// ---- Tc3_DALI_PLC_Commissioning_Tool/VISUs/Visu_DALICommissioning/Visu_Part102Scenes.TcVIS
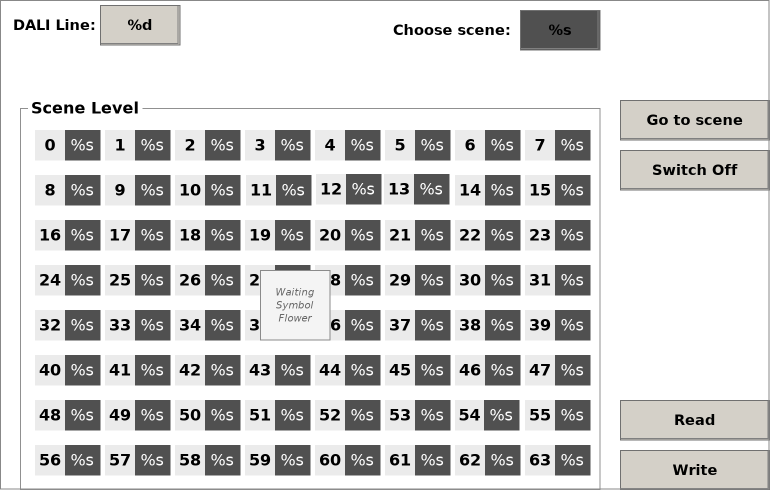
VISUALIZATION Visu_Part102Scenes  // 770x490
    GroupBox (20,100 580x390), "Scene Level"
        Group (85,30 65x30)
            Textfield (0,0 30x30), "1"
            Textfield (30,0 35x30), "%s", text variable: DALI_Commissioning.fbPart102Scenes.aScene[1], input disabled if: DALI_Commissioning.fbPart102Scenes.aNoShortAddress[1]
                p55702900: DALI_Commissioning.fbPart102Scenes.aFont[1]
                OnMouseClick: write the text variable via Default, min 0, max 255, title "Scene Value"
        Group (505,30 65x30)
            Textfield (0,0 30x30), "7"
            Textfield (30,0 35x30), "%s", text variable: DALI_Commissioning.fbPart102Scenes.aScene[7], input disabled if: DALI_Commissioning.fbPart102Scenes.aNoShortAddress[7]
                p55702900: DALI_Commissioning.fbPart102Scenes.aFont[7]
                OnMouseClick: write the text variable via Default, min 0, max 255, title "Scene Value"
        Group (435,30 65x30)
            Textfield (0,0 30x30), "6"
            Textfield (30,0 35x30), "%s", text variable: DALI_Commissioning.fbPart102Scenes.aScene[6], input disabled if: DALI_Commissioning.fbPart102Scenes.aNoShortAddress[6]
                p55702900: DALI_Commissioning.fbPart102Scenes.aFont[6]
                OnMouseClick: write the text variable via Default, min 0, max 255, title "Scene Value"
        Group (365,30 65x30)
            Textfield (0,0 30x30), "5"
            Textfield (30,0 35x30), "%s", text variable: DALI_Commissioning.fbPart102Scenes.aScene[5], input disabled if: DALI_Commissioning.fbPart102Scenes.aNoShortAddress[5]
                p55702900: DALI_Commissioning.fbPart102Scenes.aFont[5]
                OnMouseClick: write the text variable via Default, min 0, max 255, title "Scene Value"
        Group (295,30 65x30)
            Textfield (0,0 30x30), "4"
            Textfield (30,0 35x30), "%s", text variable: DALI_Commissioning.fbPart102Scenes.aScene[4], input disabled if: DALI_Commissioning.fbPart102Scenes.aNoShortAddress[4]
                p55702900: DALI_Commissioning.fbPart102Scenes.aFont[4]
                OnMouseClick: write the text variable via Default, min 0, max 255, title "Scene Value"
        Group (225,30 65x30)
            Textfield (0,0 30x30), "3"
            Textfield (30,0 35x30), "%s", text variable: DALI_Commissioning.fbPart102Scenes.aScene[3], input disabled if: DALI_Commissioning.fbPart102Scenes.aNoShortAddress[3]
                p55702900: DALI_Commissioning.fbPart102Scenes.aFont[3]
                OnMouseClick: write the text variable via Default, min 0, max 255, title "Scene Value"
        Group (155,30 65x30)
            Textfield (0,0 30x30), "2"
            Textfield (30,0 35x30), "%s", text variable: DALI_Commissioning.fbPart102Scenes.aScene[2], input disabled if: DALI_Commissioning.fbPart102Scenes.aNoShortAddress[2]
                p55702900: DALI_Commissioning.fbPart102Scenes.aFont[2]
                OnMouseClick: write the text variable via Default, min 0, max 255, title "Scene Value"
        Group (15,75 65x30)
            Textfield (0,0 30x30), "8"
            Textfield (30,0 35x30), "%s", text variable: DALI_Commissioning.fbPart102Scenes.aScene[8], input disabled if: DALI_Commissioning.fbPart102Scenes.aNoShortAddress[8]
                p55702900: DALI_Commissioning.fbPart102Scenes.aFont[8]
                OnMouseClick: write the text variable via Default, min 0, max 255, title "Scene Value"
        Group (15,120 65x30)
            Textfield (0,0 30x30), "16"
            Textfield (30,0 35x30), "%s", text variable: DALI_Commissioning.fbPart102Scenes.aScene[16], input disabled if: DALI_Commissioning.fbPart102Scenes.aNoShortAddress[16]
                p55702900: DALI_Commissioning.fbPart102Scenes.aFont[16]
                OnMouseClick: write the text variable via Default, min 0, max 255, title "Scene Value"
        Group (15,165 65x30)
            Textfield (0,0 30x30), "24"
            Textfield (30,0 35x30), "%s", text variable: DALI_Commissioning.fbPart102Scenes.aScene[24], input disabled if: DALI_Commissioning.fbPart102Scenes.aNoShortAddress[24]
                p55702900: DALI_Commissioning.fbPart102Scenes.aFont[24]
                OnMouseClick: write the text variable via Default, min 0, max 255, title "Scene Value"
        Group (15,210 65x30)
            Textfield (0,0 30x30), "32"
            Textfield (30,0 35x30), "%s", text variable: DALI_Commissioning.fbPart102Scenes.aScene[32], input disabled if: DALI_Commissioning.fbPart102Scenes.aNoShortAddress[32]
                p55702900: DALI_Commissioning.fbPart102Scenes.aFont[32]
                OnMouseClick: write the text variable via Default, min 0, max 255, title "Scene Value"
        Group (15,255 65x30)
            Textfield (0,0 30x30), "40"
            Textfield (30,0 35x30), "%s", text variable: DALI_Commissioning.fbPart102Scenes.aScene[40], input disabled if: DALI_Commissioning.fbPart102Scenes.aNoShortAddress[40]
                p55702900: DALI_Commissioning.fbPart102Scenes.aFont[40]
                OnMouseClick: write the text variable via Default, min 0, max 255, title "Scene Value"
        Group (15,300 65x30)
            Textfield (0,0 30x30), "48"
            Textfield (30,0 35x30), "%s", text variable: DALI_Commissioning.fbPart102Scenes.aScene[48], input disabled if: DALI_Commissioning.fbPart102Scenes.aNoShortAddress[48]
                p55702900: DALI_Commissioning.fbPart102Scenes.aFont[48]
                OnMouseClick: write the text variable via Default, min 0, max 255, title "Scene Value"
        Group (15,345 65x30)
            Textfield (0,0 30x30), "56"
            Textfield (30,0 35x30), "%s", text variable: DALI_Commissioning.fbPart102Scenes.aScene[56], input disabled if: DALI_Commissioning.fbPart102Scenes.aNoShortAddress[56]
                p55702900: DALI_Commissioning.fbPart102Scenes.aFont[56]
                OnMouseClick: write the text variable via Default, min 0, max 255, title "Scene Value"
        Group (85,75 65x30)
            Textfield (0,0 30x30), "9"
            Textfield (30,0 35x30), "%s", text variable: DALI_Commissioning.fbPart102Scenes.aScene[9], input disabled if: DALI_Commissioning.fbPart102Scenes.aNoShortAddress[9]
                p55702900: DALI_Commissioning.fbPart102Scenes.aFont[9]
                OnMouseClick: write the text variable via Default, min 0, max 255, title "Scene Value"
        Group (155,75 65x30)
            Textfield (0,0 30x30), "10"
            Textfield (30,0 35x30), "%s", text variable: DALI_Commissioning.fbPart102Scenes.aScene[10], input disabled if: DALI_Commissioning.fbPart102Scenes.aNoShortAddress[10]
                p55702900: DALI_Commissioning.fbPart102Scenes.aFont[10]
                OnMouseClick: write the text variable via Default, min 0, max 255, title "Scene Value"
        Group (226,75 65x30)
            Textfield (0,0 30x30), "11"
            Textfield (30,0 35x30), "%s", text variable: DALI_Commissioning.fbPart102Scenes.aScene[11], input disabled if: DALI_Commissioning.fbPart102Scenes.aNoShortAddress[11]
                p55702900: DALI_Commissioning.fbPart102Scenes.aFont[11]
                OnMouseClick: write the text variable via Default, min 0, max 255, title "Scene Value"
        Group (296,74 65x30)
            Textfield (0,0 30x30), "12"
            Textfield (30,0 35x30), "%s", text variable: DALI_Commissioning.fbPart102Scenes.aScene[12], input disabled if: DALI_Commissioning.fbPart102Scenes.aNoShortAddress[12]
                p55702900: DALI_Commissioning.fbPart102Scenes.aFont[12]
                OnMouseClick: write the text variable via Default, min 0, max 255, title "Scene Value"
        Group (364,74 65x30)
            Textfield (0,0 30x30), "13"
            Textfield (30,0 35x30), "%s", text variable: DALI_Commissioning.fbPart102Scenes.aScene[13], input disabled if: DALI_Commissioning.fbPart102Scenes.aNoShortAddress[13]
                p55702900: DALI_Commissioning.fbPart102Scenes.aFont[13]
                OnMouseClick: write the text variable via Default, min 0, max 255, title "Scene Value"
        Group (435,75 65x30)
            Textfield (0,0 30x30), "14"
            Textfield (30,0 35x30), "%s", text variable: DALI_Commissioning.fbPart102Scenes.aScene[14], input disabled if: DALI_Commissioning.fbPart102Scenes.aNoShortAddress[14]
                p55702900: DALI_Commissioning.fbPart102Scenes.aFont[14]
                OnMouseClick: write the text variable via Default, min 0, max 255, title "Scene Value"
        Group (505,75 65x30)
            Textfield (0,0 30x30), "15"
            Textfield (30,0 35x30), "%s", text variable: DALI_Commissioning.fbPart102Scenes.aScene[15], input disabled if: DALI_Commissioning.fbPart102Scenes.aNoShortAddress[15]
                p55702900: DALI_Commissioning.fbPart102Scenes.aFont[15]
                OnMouseClick: write the text variable via Default, min 0, max 255, title "Scene Value"
        Group (85,120 65x30)
            Textfield (0,0 30x30), "17"
            Textfield (30,0 35x30), "%s", text variable: DALI_Commissioning.fbPart102Scenes.aScene[17], input disabled if: DALI_Commissioning.fbPart102Scenes.aNoShortAddress[17]
                p55702900: DALI_Commissioning.fbPart102Scenes.aFont[17]
                OnMouseClick: write the text variable via Default, min 0, max 255, title "Scene Value"
        Group (155,120 65x30)
            Textfield (0,0 30x30), "18"
            Textfield (30,0 35x30), "%s", text variable: DALI_Commissioning.fbPart102Scenes.aScene[18], input disabled if: DALI_Commissioning.fbPart102Scenes.aNoShortAddress[18]
                p55702900: DALI_Commissioning.fbPart102Scenes.aFont[18]
                OnMouseClick: write the text variable via Default, min 0, max 255, title "Scene Value"
        Group (225,120 65x30)
            Textfield (0,0 30x30), "19"
            Textfield (30,0 35x30), "%s", text variable: DALI_Commissioning.fbPart102Scenes.aScene[19], input disabled if: DALI_Commissioning.fbPart102Scenes.aNoShortAddress[19]
                p55702900: DALI_Commissioning.fbPart102Scenes.aFont[19]
                OnMouseClick: write the text variable via Default, min 0, max 255, title "Scene Value"
        Group (295,120 65x30)
            Textfield (0,0 30x30), "20"
            Textfield (30,0 35x30), "%s", text variable: DALI_Commissioning.fbPart102Scenes.aScene[20], input disabled if: DALI_Commissioning.fbPart102Scenes.aNoShortAddress[20]
                p55702900: DALI_Commissioning.fbPart102Scenes.aFont[20]
                OnMouseClick: write the text variable via Default, min 0, max 255, title "Scene Value"
        Group (365,120 65x30)
            Textfield (0,0 30x30), "21"
            Textfield (30,0 35x30), "%s", text variable: DALI_Commissioning.fbPart102Scenes.aScene[21], input disabled if: DALI_Commissioning.fbPart102Scenes.aNoShortAddress[21]
                p55702900: DALI_Commissioning.fbPart102Scenes.aFont[21]
                OnMouseClick: write the text variable via Default, min 0, max 255, title "Scene Value"
        Group (435,120 65x30)
            Textfield (0,0 30x30), "22"
            Textfield (30,0 35x30), "%s", text variable: DALI_Commissioning.fbPart102Scenes.aScene[22], input disabled if: DALI_Commissioning.fbPart102Scenes.aNoShortAddress[22]
                p55702900: DALI_Commissioning.fbPart102Scenes.aFont[22]
                OnMouseClick: write the text variable via Default, min 0, max 255, title "Scene Value"
        Group (505,120 65x30)
            Textfield (0,0 30x30), "23"
            Textfield (30,0 35x30), "%s", text variable: DALI_Commissioning.fbPart102Scenes.aScene[23], input disabled if: DALI_Commissioning.fbPart102Scenes.aNoShortAddress[23]
                p55702900: DALI_Commissioning.fbPart102Scenes.aFont[23]
                OnMouseClick: write the text variable via Default, min 0, max 255, title "Scene Value"
        Group (85,165 65x30)
            Textfield (0,0 30x30), "25"
            Textfield (30,0 35x30), "%s", text variable: DALI_Commissioning.fbPart102Scenes.aScene[25], input disabled if: DALI_Commissioning.fbPart102Scenes.aNoShortAddress[25]
                p55702900: DALI_Commissioning.fbPart102Scenes.aFont[25]
                OnMouseClick: write the text variable via Default, min 0, max 255, title "Scene Value"
        Group (155,165 65x30)
            Textfield (0,0 30x30), "26"
            Textfield (30,0 35x30), "%s", text variable: DALI_Commissioning.fbPart102Scenes.aScene[26], input disabled if: DALI_Commissioning.fbPart102Scenes.aNoShortAddress[26]
                p55702900: DALI_Commissioning.fbPart102Scenes.aFont[26]
                OnMouseClick: write the text variable via Default, min 0, max 255, title "Scene Value"
        Group (225,165 65x30)
            Textfield (0,0 30x30), "27"
            Textfield (30,0 35x30), "%s", text variable: DALI_Commissioning.fbPart102Scenes.aScene[27], input disabled if: DALI_Commissioning.fbPart102Scenes.aNoShortAddress[27]
                p55702900: DALI_Commissioning.fbPart102Scenes.aFont[27]
                OnMouseClick: write the text variable via Default, min 0, max 255, title "Scene Value"
        Group (295,165 65x30)
            Textfield (0,0 30x30), "28"
            Textfield (30,0 35x30), "%s", text variable: DALI_Commissioning.fbPart102Scenes.aScene[28], input disabled if: DALI_Commissioning.fbPart102Scenes.aNoShortAddress[28]
                p55702900: DALI_Commissioning.fbPart102Scenes.aFont[28]
                OnMouseClick: write the text variable via Default, min 0, max 255, title "Scene Value"
        Group (365,165 65x30)
            Textfield (0,0 30x30), "29"
            Textfield (30,0 35x30), "%s", text variable: DALI_Commissioning.fbPart102Scenes.aScene[29], input disabled if: DALI_Commissioning.fbPart102Scenes.aNoShortAddress[29]
                p55702900: DALI_Commissioning.fbPart102Scenes.aFont[29]
                OnMouseClick: write the text variable via Default, min 0, max 255, title "Scene Value"
        Group (435,165 65x30)
            Textfield (0,0 30x30), "30"
            Textfield (30,0 35x30), "%s", text variable: DALI_Commissioning.fbPart102Scenes.aScene[30], input disabled if: DALI_Commissioning.fbPart102Scenes.aNoShortAddress[30]
                p55702900: DALI_Commissioning.fbPart102Scenes.aFont[30]
                OnMouseClick: write the text variable via Default, min 0, max 255, title "Scene Value"
        Group (505,165 65x30)
            Textfield (0,0 30x30), "31"
            Textfield (30,0 35x30), "%s", text variable: DALI_Commissioning.fbPart102Scenes.aScene[31], input disabled if: DALI_Commissioning.fbPart102Scenes.aNoShortAddress[31]
                p55702900: DALI_Commissioning.fbPart102Scenes.aFont[31]
                OnMouseClick: write the text variable via Default, min 0, max 255, title "Scene Value"
        Group (85,210 65x30)
            Textfield (0,0 30x30), "33"
            Textfield (30,0 35x30), "%s", text variable: DALI_Commissioning.fbPart102Scenes.aScene[33], input disabled if: DALI_Commissioning.fbPart102Scenes.aNoShortAddress[32]
                p55702900: DALI_Commissioning.fbPart102Scenes.aFont[33]
                OnMouseClick: write the text variable via Default, min 0, max 255, title "Scene Value"
        Group (155,210 65x30)
            Textfield (0,0 30x30), "34"
            Textfield (30,0 35x30), "%s", text variable: DALI_Commissioning.fbPart102Scenes.aScene[34], input disabled if: DALI_Commissioning.fbPart102Scenes.aNoShortAddress[34]
                p55702900: DALI_Commissioning.fbPart102Scenes.aFont[34]
                OnMouseClick: write the text variable via Default, min 0, max 255, title "Scene Value"
        Group (295,210 65x30)
            Textfield (0,0 30x30), "36"
            Textfield (30,0 35x30), "%s", text variable: DALI_Commissioning.fbPart102Scenes.aScene[36], input disabled if: DALI_Commissioning.fbPart102Scenes.aNoShortAddress[36]
                p55702900: DALI_Commissioning.fbPart102Scenes.aFont[36]
                OnMouseClick: write the text variable via Default, min 0, max 255
        Group (365,210 65x30)
            Textfield (0,0 30x30), "37"
            Textfield (30,0 35x30), "%s", text variable: DALI_Commissioning.fbPart102Scenes.aScene[37], input disabled if: DALI_Commissioning.fbPart102Scenes.aNoShortAddress[37]
                p55702900: DALI_Commissioning.fbPart102Scenes.aFont[37]
                OnMouseClick: write the text variable via Default, min 0, max 255, title "Scene Value"
        Group (435,210 65x30)
            Textfield (0,0 30x30), "38"
            Textfield (30,0 35x30), "%s", text variable: DALI_Commissioning.fbPart102Scenes.aScene[38], input disabled if: DALI_Commissioning.fbPart102Scenes.aNoShortAddress[38]
                p55702900: DALI_Commissioning.fbPart102Scenes.aFont[38]
                OnMouseClick: write the text variable via Default, min 0, max 255, title "Scene Value"
        Group (505,210 65x30)
            Textfield (0,0 30x30), "39"
            Textfield (30,0 35x30), "%s", text variable: DALI_Commissioning.fbPart102Scenes.aScene[39], input disabled if: DALI_Commissioning.fbPart102Scenes.aNoShortAddress[39]
                p55702900: DALI_Commissioning.fbPart102Scenes.aFont[39]
                OnMouseClick: write the text variable via Default, min 0, max 255, title "Scene Value"
        Group (85,255 65x30)
            Textfield (0,0 30x30), "41"
            Textfield (30,0 35x30), "%s", text variable: DALI_Commissioning.fbPart102Scenes.aScene[41], input disabled if: DALI_Commissioning.fbPart102Scenes.aNoShortAddress[41]
                p55702900: DALI_Commissioning.fbPart102Scenes.aFont[41]
                OnMouseClick: write the text variable via Default, min 0, max 255, title "Scene Value"
        Group (155,255 65x30)
            Textfield (0,0 30x30), "42"
            Textfield (30,0 35x30), "%s", text variable: DALI_Commissioning.fbPart102Scenes.aScene[42], input disabled if: DALI_Commissioning.fbPart102Scenes.aNoShortAddress[42]
                p55702900: DALI_Commissioning.fbPart102Scenes.aFont[42]
                OnMouseClick: write the text variable via Default, min 0, max 255, title "Scene Value"
        Group (225,210 65x30)
            Textfield (0,0 30x30), "35"
            Textfield (30,0 35x30), "%s", text variable: DALI_Commissioning.fbPart102Scenes.aScene[35], input disabled if: DALI_Commissioning.fbPart102Scenes.aNoShortAddress[35]
                p55702900: DALI_Commissioning.fbPart102Scenes.aFont[35]
                OnMouseClick: write the text variable via Default, min 0, max 255, title "Scene Value"
        Group (225,255 65x30)
            Textfield (0,0 30x30), "43"
            Textfield (30,0 35x30), "%s", text variable: DALI_Commissioning.fbPart102Scenes.aScene[43], input disabled if: DALI_Commissioning.fbPart102Scenes.aNoShortAddress[43]
                p55702900: DALI_Commissioning.fbPart102Scenes.aFont[43]
                OnMouseClick: write the text variable via Default, min 0, max 255, title "Scene Value"
        Group (295,255 65x30)
            Textfield (0,0 30x30), "44"
            Textfield (30,0 35x30), "%s", text variable: DALI_Commissioning.fbPart102Scenes.aScene[44], input disabled if: DALI_Commissioning.fbPart102Scenes.aNoShortAddress[44]
                p55702900: DALI_Commissioning.fbPart102Scenes.aFont[44]
                OnMouseClick: write the text variable via Default, min 0, max 255, title "Scene Value"
        Group (365,255 65x30)
            Textfield (0,0 30x30), "45"
            Textfield (30,0 35x30), "%s", text variable: DALI_Commissioning.fbPart102Scenes.aScene[45], input disabled if: DALI_Commissioning.fbPart102Scenes.aNoShortAddress[45]
                p55702900: DALI_Commissioning.fbPart102Scenes.aFont[45]
                OnMouseClick: write the text variable via Default, min 0, max 255, title "Scene Value"
        Group (435,255 65x30)
            Textfield (0,0 30x30), "46"
            Textfield (30,0 35x30), "%s", text variable: DALI_Commissioning.fbPart102Scenes.aScene[46], input disabled if: DALI_Commissioning.fbPart102Scenes.aNoShortAddress[46]
                p55702900: DALI_Commissioning.fbPart102Scenes.aFont[46]
                OnMouseClick: write the text variable via Default, min 0, max 255, title "Scene Value"
        Group (505,255 65x30)
            Textfield (0,0 30x30), "47"
            Textfield (30,0 35x30), "%s", text variable: DALI_Commissioning.fbPart102Scenes.aScene[47], input disabled if: DALI_Commissioning.fbPart102Scenes.aNoShortAddress[47]
                p55702900: DALI_Commissioning.fbPart102Scenes.aFont[47]
                OnMouseClick: write the text variable via Default, min 0, max 255, title "Scene Value"
        Group (85,300 65x30)
            Textfield (0,0 30x30), "49"
            Textfield (30,0 35x30), "%s", text variable: DALI_Commissioning.fbPart102Scenes.aScene[49], input disabled if: DALI_Commissioning.fbPart102Scenes.aNoShortAddress[49]
                p55702900: DALI_Commissioning.fbPart102Scenes.aFont[49]
                OnMouseClick: write the text variable via Default, min 0, max 255, title "Scene Value"
        Group (155,300 65x30)
            Textfield (0,0 30x30), "50"
            Textfield (30,0 35x30), "%s", text variable: DALI_Commissioning.fbPart102Scenes.aScene[50], input disabled if: DALI_Commissioning.fbPart102Scenes.aNoShortAddress[50]
                p55702900: DALI_Commissioning.fbPart102Scenes.aFont[50]
                OnMouseClick: write the text variable via Default, min 0, max 255, title "Scene Value"
        Group (225,300 65x30)
            Textfield (0,0 30x30), "51"
            Textfield (30,0 35x30), "%s", text variable: DALI_Commissioning.fbPart102Scenes.aScene[51], input disabled if: DALI_Commissioning.fbPart102Scenes.aNoShortAddress[51]
                p55702900: DALI_Commissioning.fbPart102Scenes.aFont[51]
                OnMouseClick: write the text variable via Default, min 0, max 255, title "Scene Value"
        Group (295,300 65x30)
            Textfield (0,0 30x30), "52"
            Textfield (30,0 35x30), "%s", text variable: DALI_Commissioning.fbPart102Scenes.aScene[52], input disabled if: DALI_Commissioning.fbPart102Scenes.aNoShortAddress[52]
                p55702900: DALI_Commissioning.fbPart102Scenes.aFont[52]
                OnMouseClick: write the text variable via Default, min 0, max 255, title "Scene Value"
        Group (365,300 65x30)
            Textfield (0,0 30x30), "53"
            Textfield (30,0 35x30), "%s", text variable: DALI_Commissioning.fbPart102Scenes.aScene[53], input disabled if: DALI_Commissioning.fbPart102Scenes.aNoShortAddress[53]
                p55702900: DALI_Commissioning.fbPart102Scenes.aFont[53]
                OnMouseClick: write the text variable via Default, min 0, max 255, title "Scene Value"
        Group (435,300 64x30)
            Textfield (0,0 29x30), "54"
            Textfield (29,0 35x30), "%s", text variable: DALI_Commissioning.fbPart102Scenes.aScene[54], input disabled if: DALI_Commissioning.fbPart102Scenes.aNoShortAddress[54]
                p55702900: DALI_Commissioning.fbPart102Scenes.aFont[54]
                OnMouseClick: write the text variable via Default, min 0, max 255, title "Scene Value"
        Group (505,300 65x30)
            Textfield (0,0 30x30), "55"
            Textfield (30,0 35x30), "%s", text variable: DALI_Commissioning.fbPart102Scenes.aScene[55], input disabled if: DALI_Commissioning.fbPart102Scenes.aNoShortAddress[55]
                p55702900: DALI_Commissioning.fbPart102Scenes.aFont[55]
                OnMouseClick: write the text variable via Default, min 0, max 255, title "Scene Value"
        Group (85,345 65x30)
            Textfield (0,0 30x30), "57"
            Textfield (30,0 35x30), "%s", text variable: DALI_Commissioning.fbPart102Scenes.aScene[57], input disabled if: DALI_Commissioning.fbPart102Scenes.aNoShortAddress[57]
                p55702900: DALI_Commissioning.fbPart102Scenes.aFont[57]
                OnMouseClick: write the text variable via Default, min 0, max 255, title "Scene Value"
        Group (155,345 65x30)
            Textfield (0,0 30x30), "58"
            Textfield (30,0 35x30), "%s", text variable: DALI_Commissioning.fbPart102Scenes.aScene[58], input disabled if: DALI_Commissioning.fbPart102Scenes.aNoShortAddress[58]
                p55702900: DALI_Commissioning.fbPart102Scenes.aFont[58]
                OnMouseClick: write the text variable via Default, min 0, max 255, title "Scene Value"
        Group (225,345 65x30)
            Textfield (0,0 30x30), "59"
            Textfield (30,0 35x30), "%s", text variable: DALI_Commissioning.fbPart102Scenes.aScene[59], input disabled if: DALI_Commissioning.fbPart102Scenes.aNoShortAddress[59]
                p55702900: DALI_Commissioning.fbPart102Scenes.aFont[59]
                OnMouseClick: write the text variable via Default, min 0, max 255, title "Scene Value"
        Group (295,345 65x30)
            Textfield (0,0 30x30), "60"
            Textfield (30,0 35x30), "%s", text variable: DALI_Commissioning.fbPart102Scenes.aScene[60], input disabled if: DALI_Commissioning.fbPart102Scenes.aNoShortAddress[60]
                p55702900: DALI_Commissioning.fbPart102Scenes.aFont[60]
                OnMouseClick: write the text variable via Default, min 0, max 255, title "Scene Value"
        Group (365,345 65x30)
            Textfield (0,0 30x30), "61"
            Textfield (30,0 35x30), "%s", text variable: DALI_Commissioning.fbPart102Scenes.aScene[61], input disabled if: DALI_Commissioning.fbPart102Scenes.aNoShortAddress[61]
                p55702900: DALI_Commissioning.fbPart102Scenes.aFont[61]
                OnMouseClick: write the text variable via Default, min 0, max 255, title "Scene Value"
        Group (435,345 65x30)
            Textfield (0,0 30x30), "62"
            Textfield (30,0 35x30), "%s", text variable: DALI_Commissioning.fbPart102Scenes.aScene[62], input disabled if: DALI_Commissioning.fbPart102Scenes.aNoShortAddress[62]
                p55702900: DALI_Commissioning.fbPart102Scenes.aFont[62]
                OnMouseClick: write the text variable via Default, min 0, max 255, title "Scene Value"
        Group (505,345 65x30)
            Textfield (0,0 30x30), "63"
            Textfield (30,0 35x30), "%s", text variable: DALI_Commissioning.fbPart102Scenes.aScene[63], input disabled if: DALI_Commissioning.fbPart102Scenes.aNoShortAddress[63]
                p55702900: DALI_Commissioning.fbPart102Scenes.aFont[63]
                OnMouseClick: write the text variable via Default, min 0, max 255, title "Scene Value"
        WaitingSymbolFlower (240,170 70x70), invisible if: DALI_Commissioning.fbPart102Scenes.bHideWaitSymbol
        Group (15,30 65x30)
            Textfield (0,0 30x30), "0"
            Textfield (30,0 35x30), "%s", text variable: DALI_Commissioning.fbPart102Scenes.aScene[0], input disabled if: DALI_Commissioning.fbPart102Scenes.aNoShortAddress[0]
                p55702900: DALI_Commissioning.fbPart102Scenes.aFont[0]
                OnMouseClick: write the text variable via Default, min 0, max 255, title "Scene Value"
    Button (620,400 150x40), "Read"
        OnMouseClick: execute { DALI_Commissioning.fbPart102Scenes.bRead := TRUE; }
    Button (620,450 150x40), "Write"
        OnMouseClick: execute { DALI_Commissioning.fbPart102Scenes.bWrite := TRUE; }
    Button (620,100 150x40), "Go to scene"
        OnMouseClick: execute { DALI_Commissioning.fbPart102Scenes.bGoToScene := TRUE; }
    Button (620,150 150x40), "Switch Off"
        OnMouseClick: execute { DALI_Commissioning.fbPart102Scenes.bSwitchOff := TRUE; }
    Textfield (390,10 120x40), "Choose scene:"
    Button (520,10 80x40), "%s", text variable: DALI_Commissioning.fbPart102Scenes.nScene
        OnMouseClick: write the text variable via Default, min 0, max 15, title "Choose scene"
    Group (10,5 170x40)
        Textfield (0,0 110x40), "DALI Line:"
        Button (90,0 80x40), "%d", text variable: GVL_Internal.nDALILine
            OnMouseClick: write the text variable via Default, min 1, max GVL_Internal.nNumberOfDALI_Lines, title "Choose line"
END_VISUALIZATION

// ---- Tc3_DALI_PLC_Commissioning_Tool/VISUs/Visu_DALICommissioning/Visu_Part102SetFading.TcVIS
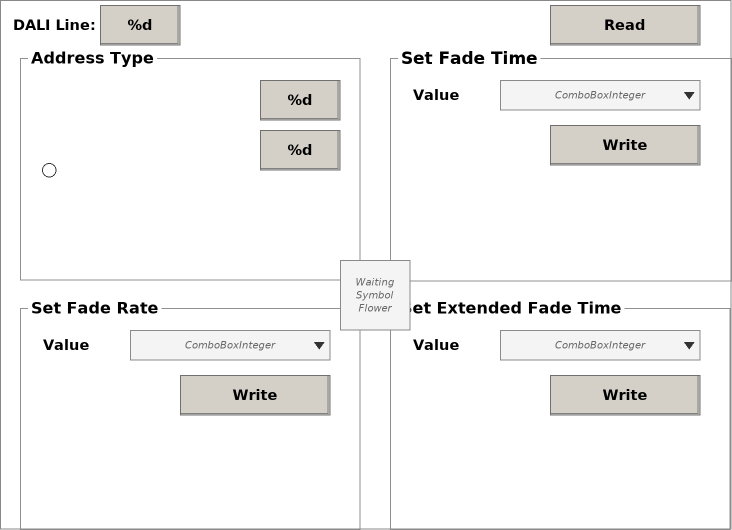
VISUALIZATION Visu_Part102SetFading  // 732x530
    GroupBox (390,50 342x231), "Set Fade Time"
        Textfield (20,30 100x30), "Value"
        ComboBoxInteger (110,30 200x30), variable: DALI_Commissioning.fbPart102SetFading.eFadeTime, text list: 'FadeTime'
        Button (160,75 150x40), "Write"
            OnMouseClick: execute { DALI_Commissioning.fbPart102SetFading.bWriteFadeTime := TRUE; }
    GroupBox (20,50 340x230), "Address Type"
        Button (240,30 80x40), "%d", text variable: DALI_Commissioning.fbPart102SetFading.nShortAddress
            OnMouseClick: write the text variable via Default, min 0, max 63, title "Insert Short Address"
        RadioButton (20,20 190x200), variable: DALI_Commissioning.fbPart102SetFading.eAddressType
            Areas[0]: Text=Short Address
            Areas[1]: Text=Group Address
            Areas[2]: Text=Broadcast
            Areas[3]: Text=Unaddressed
        Button (240,80 80x40), "%d", text variable: DALI_Commissioning.fbPart102SetFading.nGroupAddress
            OnMouseClick: write the text variable via Default, min 0, max 15, title "Insert Group Address"
    GroupBox (20,300 340x230), "Set Fade Rate"
        Textfield (20,30 100x30), "Value"
        ComboBoxInteger (110,30 200x30), variable: DALI_Commissioning.fbPart102SetFading.eFadeRate, text list: 'FadeRate'
        Button (160,75 150x40), "Write"
            OnMouseClick: execute { DALI_Commissioning.fbPart102setFading.bWriteFadeRate := TRUE; }
    GroupBox (390,300 340x230), "Set Extended Fade Time"
        Textfield (20,30 100x30), "Value"
        ComboBoxInteger (110,30 200x30), tooltip "Extended Fade Time only valid if Fade Time equals 0!", variable: DALI_Commissioning.fbPart102SetFading.eExtendedFadeTime, input disabled if: DALI_Commissioning.fbPart102SetFading.bNoFadeTime, text list: 'ExtendedFadeTime'
        Button (160,75 150x40), "Write", tooltip "Extended Fade Time only valid if Fade Time equals 0!", invisible if: DALI_Commissioning.fbPart102SetFading.bNoFadeTime, input disabled if: DALI_Commissioning.fbPart102SetFading.bNoFadeTime
            OnMouseClick: execute { DALI_Commissioning.fbPart102SetFading.bWriteExtendedFadeTime:=true; }
    Button (550,5 150x40), "Read", tooltip "Reads all Fading Parameters", invisible if: ( DALI_Commissioning.fbPart102SetFading.eAddressType >=1), input disabled if: ( DALI_Commissioning.fbPart102SetFading.eAddressType >=1)
        OnMouseClick: execute { DALI_Commissioning.fbPart102SetFading.bRead := TRUE; }
    WaitingSymbolFlower (340,260 70x70), invisible if: DALI_Commissioning.fbPart102SetFading.bHideWaitSymbol
    Group (10,5 170x40)
        Textfield (0,0 110x40), "DALI Line:"
        Button (90,0 80x40), "%d", text variable: GVL_Internal.nDALILine
            OnMouseClick: write the text variable via Default, min 1, max GVL_Internal.nNumberOfDALI_Lines, title "Choose line"
END_VISUALIZATION

// ---- Tc3_DALI_PLC_Commissioning_Tool/VISUs/Visu_DALICommissioning/Visu_Part103Addressing.TcVIS
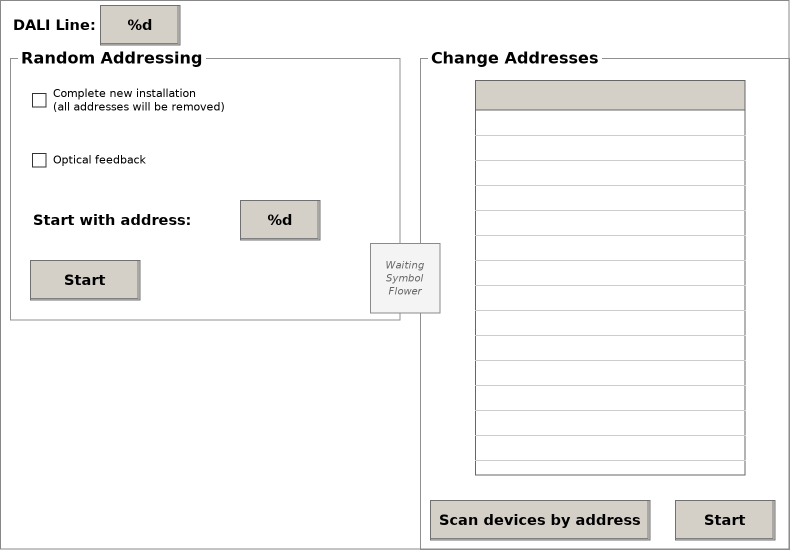
VISUALIZATION Visu_Part103Addressing  // 790x550
    GroupBox (420,50 370x500), "Change Addresses"
        Table (55,30 270x395), data array: DALI_Commissioning.fbPart103Addressing.aChangeAddressList
            p3854506369: DALI_Commissioning.fbPart103Addressing.aChangeAddressList[INDEX].nOldAddress
            p1892666644: DALI_Commissioning.fbPart103Addressing.aChangeAddressList[INDEX].nNewAddress
            p338671338: DALI_Commissioning.fbPart103Addressing.aChangeAddressList[INDEX].nRandomAddress
            p2170511999: DALI_Commissioning.fbPart103Addressing.aChangeAddressList[INDEX].nErrors
            Columns.Column.[0].Template: DALI_Commissioning.fbPart103Addressing.aNoShortAddress[INDEX]
            Columns.Column.[1].Template: DALI_Commissioning.fbPart103Addressing.aNoShortAddress[INDEX]; OnMouseClick: write the text variable via Default, min 0, max 63, title "New Short Address"
        Button (255,450 100x40), "Start"
            OnMouseClick: execute { DALI_Commissioning.fbPart103Addressing.bStartChangeAddress := TRUE; }
        Button (10,450 220x40), "Scan devices by address"
            OnMouseClick: execute { DALI_Commissioning.fbPart103Addressing.bScanDevices := TRUE; }
    GroupBox (10,50 390x270), "Random Addressing"
        Button (20,210 110x40), "Start"
            OnMouseClick: execute { DALI_Commissioning.fbPart103Addressing.bStartRandomAddressing := TRUE; }
        Checkbox (20,30 360x40), "Complete new installation (all addresses will be removed)", variable: DALI_Commissioning.fbPart103Addressing.bNewInstallation
        Checkbox (20,90 360x40), "Optical feedback", variable: DALI_Commissioning.fbPart103Addressing.bOpticalFeedback
        Textfield (20,150 200x40), "Start with address:"
        Button (230,150 80x40), "%d", text variable: DALI_Commissioning.fbPart103Addressing.nStartAddress
            OnMouseClick: write DALI_Commissioning.fbPart103Addressing.nStartAddress via Default, min 0, max 63, title "Insert Short Address"
    WaitingSymbolFlower (370,243 70x70), invisible if: DALI_Commissioning.fbPart103Addressing.bHideWaitSymbol
    Group (10,5 170x40)
        Textfield (0,0 110x40), "DALI Line:"
        Button (90,0 80x40), "%d", text variable: GVL_Internal.nDALILine
            OnMouseClick: write the text variable via Default, min 1, max GVL_Internal.nNumberOfDALI_Lines, title "Choose line"
END_VISUALIZATION

// ---- Tc3_DALI_PLC_Commissioning_Tool/VISUs/Visu_DALICommissioning/Visu_Part103MemoryBank.TcVIS
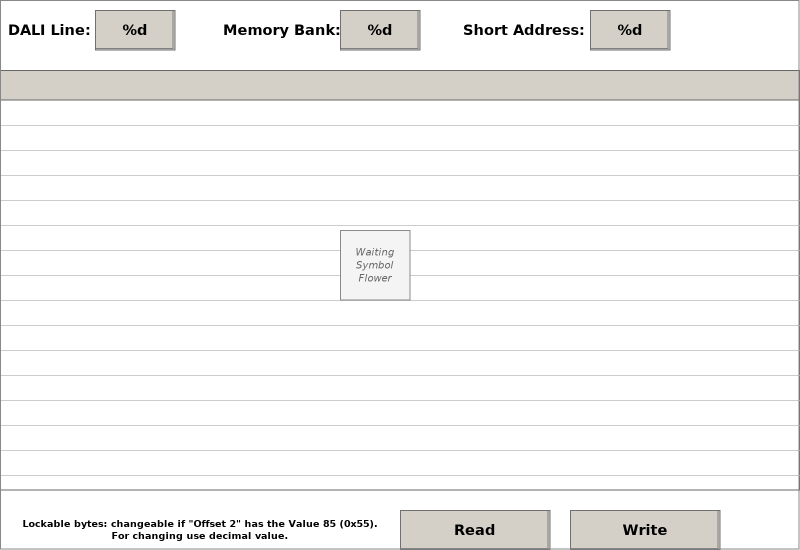
VISUALIZATION Visu_Part103MemoryBank  // 800x550
    Table (0,70 800x420), data array: DALI_Commissioning.fbPart103MemoryPages.aMemoryBank
        p3854506369: DALI_Commissioning.fbPart103MemoryPages.aMemoryBank[INDEX].sOffset
        p1892666644: DALI_Commissioning.fbPart103MemoryPages.aMemoryBank[INDEX].sName
        p338671338: DALI_Commissioning.fbPart103MemoryPages.aMemoryBank[INDEX].nValueDec
        p2170511999: DALI_Commissioning.fbPart103MemoryPages.aMemoryBank[INDEX].nValueHex
        p1755163831: Value Dec
        p4092479075: Value Hex
        p1137915858: DALI_Commissioning.fbPart103MemoryPages.nOffset
        Columns.Column.[0].Template: DALI_Commissioning.fbPart103MemoryPages.aNoValue[INDEX]
        Columns.Column.[1].Template: DALI_Commissioning.fbPart103MemoryPages.aNoValue[INDEX]
        Columns.Column.[2].Template: DALI_Commissioning.fbPart103MemoryPages.aNoValue[INDEX]; DALI_Commissioning.fbPart103MemoryPages.nMemoryBank=0; OnMouseClick: write the text variable via Default, min 0, max 255, title "Lockable variable decimal"
        Columns.Column.[3].Template: DALI_Commissioning.fbPart103MemoryPages.aNoValue[INDEX]; OnMouseClick: write the text variable via Default, title "Lockable variable hexadecimal"
    Button (400,510 150x40), "Read"
        OnMouseClick: execute { DALI_Commissioning.fbPart103MemoryPages.bRead := TRUE; }
    Button (570,510 150x40), "Write"
        OnMouseClick: execute { DALI_Commissioning.fbPart103MemoryPages.bWrite := TRUE; }
    Textfield (15,510 370x40), "Lockable bytes: changeable if "Offset 2" has the Value 85 (0x55). For changing use decimal value."
    WaitingSymbolFlower (340,230 70x70), invisible if: DALI_Commissioning.fbPart103MemoryPages.bHideWaitSymbol
    Textfield (460,10 130x40), "Short Address:"
    Button (590,10 80x40), "%d", text variable: DALI_Commissioning.fbPart103MemoryPages.nAddress
        OnMouseClick: write the text variable via Default, min 0, max 63, title "Insert Short Address"
    Group (220,10 200x40)
        Textfield (0,0 150x40), "Memory Bank:"
        Button (120,0 80x40), "%d", text variable: DALI_Commissioning.fbPart103MemoryPages.nMemoryBank
            OnMouseClick: write the text variable via Default, min 0, max 255, title "Insert Memory Bank"
    Group (5,10 170x40)
        Textfield (0,0 110x40), "DALI Line:"
        Button (90,0 80x40), "%d", text variable: GVL_Internal.nDALILine
            OnMouseClick: write the text variable via Default, min 1, max GVL_Internal.nNumberOfDALI_Lines, title "Choose line"
END_VISUALIZATION

// ---- Tc3_DALI_PLC_Commissioning_Tool/VISUs/Visu_DALICommissioning/Visu_Part103Parameters.TcVIS
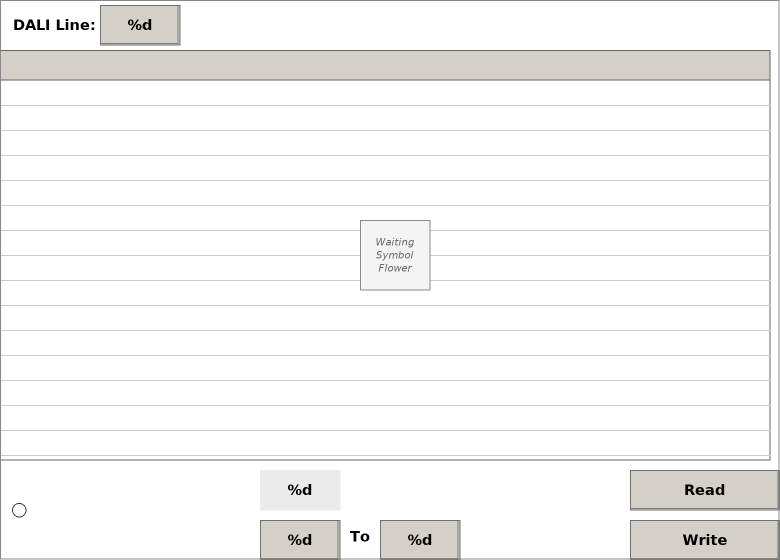
VISUALIZATION Visu_Part103Parameters  // 780x560
    Table (0,50 770x410), data array: DALI_Commissioning.fbPart103Parameters.aParameters
        p1137915858: DALI_Commissioning.fbPart103Parameters.nSelectedAddress
        p3854506369: DALI_Commissioning.fbPart103Parameters.aParameters[INDEX].nOperatingMode
        p1892666644: DALI_Commissioning.fbPart103Parameters.aParameters[INDEX].sInstanceType0
        p338671338: DALI_Commissioning.fbPart103Parameters.aParameters[INDEX].sInstanceType1
        p2170511999: DALI_Commissioning.fbPart103Parameters.aParameters[INDEX].sInstanceType2
        p3723444502: DALI_Commissioning.fbPart103Parameters.aParameters[INDEX].sInstanceType3
        p1218418051: DALI_Commissioning.fbPart103Parameters.aParameters[INDEX].sInstanceType4
        p511219082: IT0 (Generic Input)
        p1755163831: IT1 (PushButton)
        p4092479075: IT2 (Absolute Input)
        p2237128397: IT3 (Occupancy)
        p505689113: IT4 (Light Sensor)
        Columns.Column.[0].Template: OnMouseClick: write the text variable via Default, min 0, max 255, title "Insert Operating Mode 0, 128-255"
    RadioButton (10,460 230x100), variable: DALI_Commissioning.fbPart103Parameters.nAddressRange
        Areas[0]: Text=Single Short Address
        Areas[1]: Text=Short Address Range
    Textfield (260,470 80x40), "%d", text variable: DALI_Commissioning.fbPart103Parameters.nSelectedAddress
    Button (260,520 80x40), "%d", text variable: DALI_Commissioning.fbPart103Parameters.nStartAddress
        OnMouseClick: write the text variable via Default, min 0, max 63, title "Insert Short Address"
    Button (380,520 80x40), "%d", text variable: DALI_Commissioning.fbPart103Parameters.nEndAddress
        OnMouseClick: write the text variable via Default, min 0, max 63, title "Insert Short Address"
    Button (630,470 150x40), "Read"
        OnMouseClick: execute { DALI_Commissioning.fbPart103Parameters.bRead := true; }
    Button (630,520 150x40), "Write"
        OnMouseClick: execute { DALI_Commissioning.fbPart103Parameters.bWrite := true; }
    Textfield (335,521 50x31), "To"
    WaitingSymbolFlower (360,220 70x70), invisible if: DALI_Commissioning.fbPart103Parameters.bHideWaitSymbol
    Group (10,5 170x40)
        Textfield (0,0 110x40), "DALI Line:"
        Button (90,0 80x40), "%d", text variable: GVL_Internal.nDALILine
            OnMouseClick: write the text variable via Default, min 1, max GVL_Internal.nNumberOfDALI_Lines, title "Choose line"
END_VISUALIZATION

// ---- Tc3_DALI_PLC_Commissioning_Tool/VISUs/Visu_DALICommissioning/Visu_Part207Parameters.TcVIS
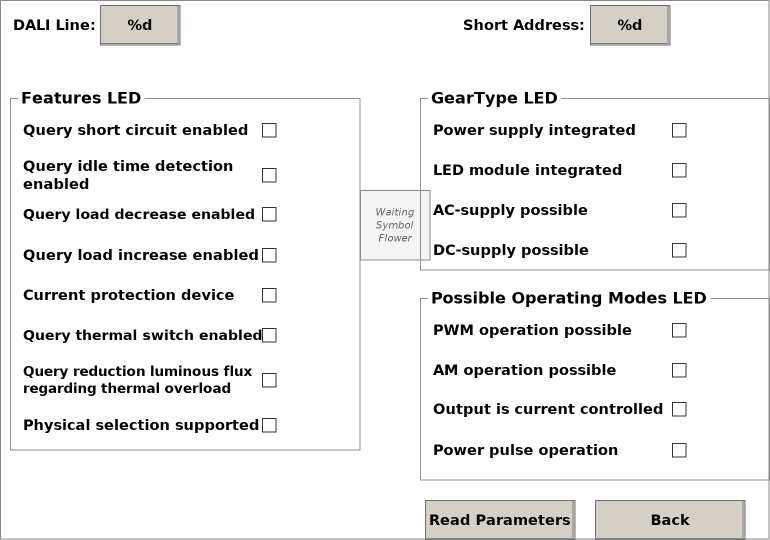
VISUALIZATION Visu_Part207Parameters  // 770x540
    Button (425,500 150x40), "Read Parameters"
        OnMouseClick: execute { DALI_Commissioning.fbPart207ParametersLED.bRead:=TRUE; }
    WaitingSymbolFlower (360,190 70x70), invisible if: DALI_Commissioning.fbPart207ParametersLED.bHideWaitSymbol
    GroupBox (420,90 350x180), "GearType LED"
        Textfield (10,25 220x30), "Power supply integrated"
        Checkbox (250,25 30x30), variable: DALI_Commissioning.fbPart207ParametersLED.bLEDPowerSupply
        Textfield (10,65 170x30)
        Textfield (10,65 220x30), "LED module integrated"
        Textfield (10,145 220x30), "DC-supply possible"
        Textfield (10,105 220x30), "AC-supply possible"
        Checkbox (250,65 30x30), variable: DALI_Commissioning.fbPart207ParametersLED.bLEDModule
        Checkbox (250,145 30x30), variable: DALI_Commissioning.fbPart207ParametersLED.bDCSupply
        Checkbox (250,105 30x30), variable: DALI_Commissioning.fbPart207ParametersLED.bACSupply
    GroupBox (10,90 350x360), "Features LED"
        Textfield (10,25 240x30), "Query short circuit enabled"
        Checkbox (250,25 30x30), variable: DALI_Commissioning.fbPart207ParametersLED.bQueryShortCircuitEnabled
        Textfield (10,65 240x30)
        Textfield (10,65 240x40), "Query idle time detection enabled"
        Textfield (10,150 240x30), "Query load increase enabled"
        Textfield (10,109 240x30), "Query load decrease enabled"
        Checkbox (250,70 30x30), variable: DALI_Commissioning.fbPart207ParametersLED.bQueryIdleTimeDetectionEnabled
        Checkbox (250,150 30x30), variable: DALI_Commissioning.fbPart207ParametersLED.bQueryLoadIncreaseEnabled
        Checkbox (250,109 30x30), variable: DALI_Commissioning.fbPart207ParametersLED.bQueryLoadDecreaseEnabled
        Textfield (10,190 240x30), "Current protection device"
        Checkbox (250,190 30x30), variable: DALI_Commissioning.fbPart207ParametersLED.bQueryCurrentProtectionDevicePresent
        Checkbox (250,230 30x30), variable: DALI_Commissioning.fbPart207ParametersLED.bQueryThermalSwitchEnabled
        Checkbox (250,275 30x30), variable: DALI_Commissioning.fbPart207ParametersLED.bQueryReductionOfLuminouFluxRegardingThermalOverloadEnabled
        Checkbox (250,320 30x30), variable: DALI_Commissioning.fbPart207ParametersLED.bPhysicalSelectionSupported
        Textfield (10,230 240x30), "Query thermal switch enabled"
        Textfield (10,270 240x40), "Query reduction luminous flux regarding thermal overload"
        Textfield (10,320 240x30), "Physical selection supported"
    Button (595,500 150x40), "Back"
        OnMouseClick: change screen: Previous 
    Group (460,5 210x40)
        Textfield (0,0 130x40), "Short Address:"
        Button (130,0 80x40), "%d", text variable: DALI_Commissioning.fbPart207ParametersLED.nAddress
            OnMouseClick: write the text variable via Default, min 0, max 63, title "Insert Short Address"
    Group (10,5 170x40)
        Textfield (0,0 110x40), "DALI Line:"
        Button (90,0 80x40), "%d", text variable: GVL_Internal.nDALILine
            OnMouseClick: write the text variable via Default, min 1, max GVL_Internal.nNumberOfDALI_Lines, title "Choose line"
    GroupBox (420,290 350x190), "Possible Operating Modes LED", invisible if: DALI_Commissioning.fbPart207ParametersLED.bInvisible
        Checkbox (250,25 30x30), variable: DALI_Commissioning.fbPart207ParametersLED.bPWMOperation
        Textfield (10,65 240x30)
        Textfield (10,65 240x30), "AM operation possible"
        Textfield (10,145 240x30), "Power pulse operation"
        Textfield (10,104 240x30), "Output is current controlled"
        Checkbox (250,65 30x30), variable: DALI_Commissioning.fbPart207ParametersLED.bAMOperation
        Checkbox (250,145 30x30), variable: DALI_Commissioning.fbPart207ParametersLED.bPowerPulseOperation
        Checkbox (250,104 30x30), variable: DALI_Commissioning.fbPart207ParametersLED.bOutputCurrentControlled
        Textfield (10,25 240x30), "PWM operation possible"
END_VISUALIZATION

// ---- Tc3_DALI_PLC_Commissioning_Tool/VISUs/Visu_DALICommissioning/Visu_Part207Status.TcVIS
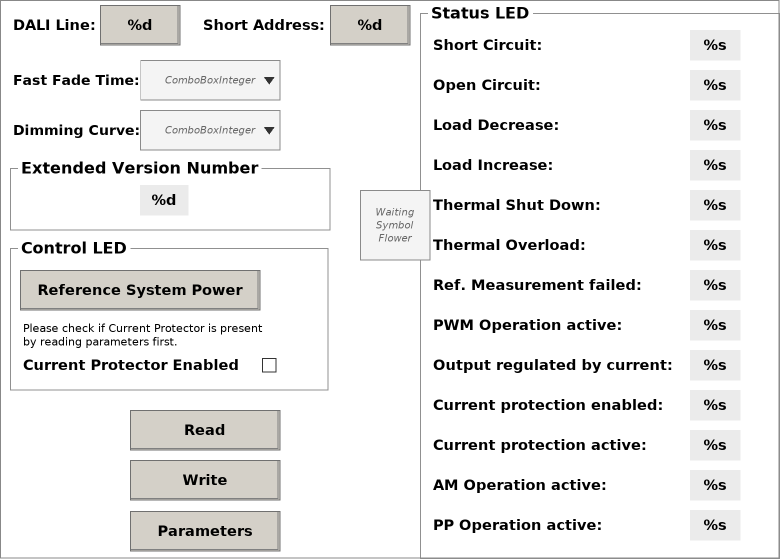
VISUALIZATION Visu_Part207Status  // 780x559
    GroupBox (420,5 360x554), "Status LED"
        Textfield (10,25 250x30), "Short Circuit:"
        Textfield (10,65 250x30), "Open Circuit:"
        Textfield (10,105 250x30), "Load Decrease:"
        Textfield (270,25 50x30), "%s", text variable: DALI_Commissioning.fbPart207StatusLED.sShortCircuit
        Textfield (270,65 50x30), "%s", text variable: DALI_Commissioning.fbPart207StatusLED.sOpenCircuit
        Textfield (270,105 50x30), "%s", text variable: DALI_Commissioning.fbPart207StatusLED.sLoadDecrease
        Textfield (10,145 250x30), "Load Increase:"
        Textfield (270,145 50x30), "%s", text variable: DALI_Commissioning.fbPart207StatusLED.sLoadIncrease
        Textfield (10,345 250x30), "Output regulated by current:", invisible if: DALI_Commissioning.fbPart207StatusLED.bInvisible
        Textfield (10,385 250x30), "Current protection enabled:", invisible if: DALI_Commissioning.fbPart207StatusLED.bInvisible
        Textfield (10,425 250x30), "Current protection active:", invisible if: DALI_Commissioning.fbPart207StatusLED.bInvisible
        Textfield (10,185 250x30), "Thermal Shut Down:"
        Textfield (10,225 250x30), "Thermal Overload:"
        Textfield (10,265 250x30), "Ref. Measurement failed:"
        Textfield (10,465 250x30), "AM Operation active:", invisible if: DALI_Commissioning.fbPart207StatusLED.bInvisible
        Textfield (10,505 250x30), "PP Operation active:", invisible if: DALI_Commissioning.fbPart207StatusLED.bInvisible
        Textfield (10,305 250x30), "PWM Operation active:", invisible if: DALI_Commissioning.fbPart207StatusLED.bInvisible
        Textfield (270,225 50x30), "%s", text variable: DALI_Commissioning.fbPart207StatusLED.sThermalOverload
        Textfield (270,425 50x30), "%s", text variable: DALI_Commissioning.fbPart207StatusLED.sCurrentProtectorActive, invisible if: DALI_Commissioning.fbPart207StatusLED.bInvisible
        Textfield (270,385 50x30), "%s", text variable: DALI_Commissioning.fbPart207StatusLED.sCurrentProtectorEnabled, invisible if: DALI_Commissioning.fbPart207StatusLED.bInvisible
        Textfield (270,345 50x30), "%s", text variable: DALI_Commissioning.fbPart207StatusLED.sOutputCurrentControlled, invisible if: DALI_Commissioning.fbPart207StatusLED.bInvisible
        Textfield (270,465 50x30), "%s", text variable: DALI_Commissioning.fbPart207StatusLED.sAMOperation, invisible if: DALI_Commissioning.fbPart207StatusLED.bInvisible
        Textfield (270,505 50x30), "%s", text variable: DALI_Commissioning.fbPart207StatusLED.sPowerPulseOperation, invisible if: DALI_Commissioning.fbPart207StatusLED.bInvisible
        Textfield (270,265 50x30), "%s", text variable: DALI_Commissioning.fbPart207StatusLED.sReferenceMeasurementFailed
        Textfield (270,185 50x30), "%s", text variable: DALI_Commissioning.fbPart207StatusLED.sThermalShutDown
        Textfield (270,305 50x30), "%s", text variable: DALI_Commissioning.fbPart207StatusLED.sPWMOperation, invisible if: DALI_Commissioning.fbPart207StatusLED.bInvisible
    Button (130,460 150x40), "Write"
        OnMouseClick: execute { DALI_Commissioning.fbPart207StatusLED.bWrite := TRUE; }
    GroupBox (10,240 318x150), "Control LED"
        Textfield (10,110 230x30), "Current Protector Enabled", invisible if: NOT DALI_Commissioning.fbPart207ParametersLED.bQueryCurrentProtectionDevicePresent
        Checkbox (250,110 30x30), variable: DALI_Commissioning.fbPart207StatusLED.bCurrentProtector, invisible if: NOT DALI_Commissioning.fbPart207ParametersLED.bQueryCurrentProtectionDevicePresent, input disabled if: DALI_Commissioning.fbPart207ParametersLED.bQueryCurrentProtectionDevicePresent
        Button (10,30 240x40), "Reference System Power"
            OnMouseClick: execute { DALI_Commissioning.fbPart207StatusLED.bReferenceSystempower := TRUE; }
        Label (10,80 300x30), "Please check if Current Protector is present by reading parameters first."
    Button (130,410 150x40), "Read"
        OnMouseClick: execute { DALI_Commissioning.fbPart207StatusLED.bRead := TRUE; }
    WaitingSymbolFlower (360,190 70x70), invisible if: DALI_Commissioning.fbPart207StatusLED.bHideWaitSymbol
    GroupBox (10,160 320x70), "Extended Version Number"
        Textfield (130,25 48x30), "%d", text variable: DALI_Commissioning.fbPart207StatusLED.nExtendedVersionNumber
    Button (130,511 150x40), "Parameters"
        OnMouseClick: change screen: Visu_Part207Parameters
    Group (200,5 210x40)
        Textfield (0,0 130x40), "Short Address:"
        Button (130,0 80x40), "%d", text variable: DALI_Commissioning.fbPart207StatusLED.nAddress
            OnMouseClick: write the text variable via Default, min 0, max 63, title "Insert Short Address"
    Group (10,110 270x40)
        Textfield (0,0 130x40), "Dimming Curve:"
        ComboBoxInteger (130,0 140x40), variable: DALI_Commissioning.fbPart207StatusLED.eDimmingCurve, text list: 'DimmingCurve'
    Group (10,60 270x40)
        ComboBoxInteger (130,0 140x40), variable: DALI_Commissioning.fbPart207StatusLED.eFastFadeTime, text list: 'FastFadeTime'
        Textfield (0,0 130x40), "Fast Fade Time:"
    Group (10,5 170x40)
        Textfield (0,0 110x40), "DALI Line:"
        Button (90,0 80x40), "%d", text variable: GVL_Internal.nDALILine
            OnMouseClick: write the text variable via Default, min 1, max GVL_Internal.nNumberOfDALI_Lines, title "Choose line"
END_VISUALIZATION

// ---- Tc3_DALI_PLC_Commissioning_Tool/VISUs/Visu_DALICommissioning/Visu_Part300GenericDevice.TcVIS
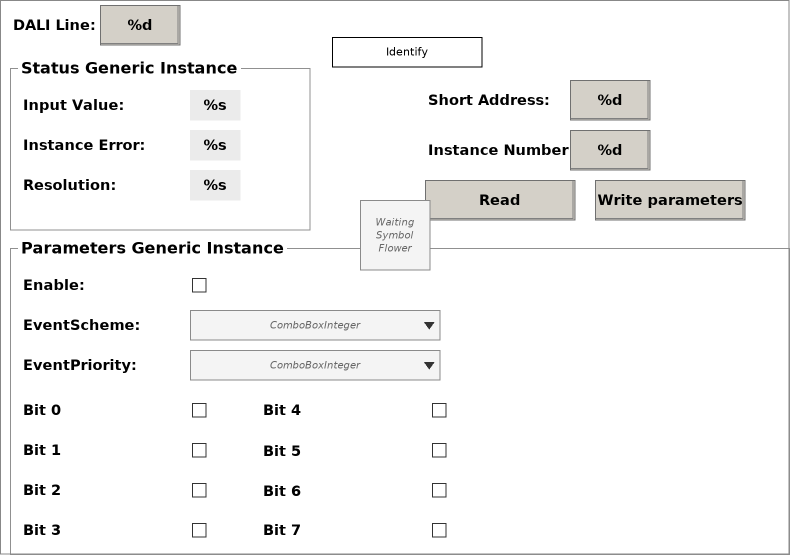
VISUALIZATION Visu_Part300GenericDevice  // 790x555
    GroupBox (10,240 780x315), "Parameters Generic Instance"
        Textfield (10,30 150x30), "Enable:"
        Checkbox (180,30 30x30), variable: DALI_Commissioning.fbPart300GenericDevice.bEnable
        Textfield (10,110 150x30), "EventPriority:"
        Textfield (10,195 100x30), "Bit 1"
        Textfield (10,155 100x30), "Bit 0"
        Checkbox (180,155 30x30), variable: DALI_Commissioning.fbPart300GenericDevice.bBit0
        Checkbox (180,195 30x30), variable: DALI_Commissioning.fbPart300GenericDevice.bBit1
        Textfield (10,235 100x30), "Bit 2"
        Textfield (250,155 100x30), "Bit 4"
        Textfield (250,196 100x30), "Bit 5"
        Checkbox (420,195 30x30), variable: DALI_Commissioning.fbPart300GenericDevice.bBit5
        Checkbox (420,155 30x30), variable: DALI_Commissioning.fbPart300GenericDevice.bBit4
        Checkbox (180,275 30x30), variable: DALI_Commissioning.fbPart300GenericDevice.bBit3
        Checkbox (180,235 30x30), variable: DALI_Commissioning.fbPart300GenericDevice.bBit2
        ComboBoxInteger (180,70 250x30), variable: DALI_Commissioning.fbPart300GenericDevice.eEventScheme, text list: 'EventScheme'
        Textfield (10,70 150x30), "EventScheme:"
        Textfield (250,236 100x30), "Bit 6"
        ComboBoxInteger (180,110 250x30), variable: DALI_Commissioning.fbPart300GenericDevice.eEventPriority, text list: 'EventPriority'
        Textfield (10,275 100x30), "Bit 3"
        Checkbox (420,235 30x30), variable: DALI_Commissioning.fbPart300GenericDevice.bBit6
        Checkbox (420,275 30x30), variable: DALI_Commissioning.fbPart300GenericDevice.bBit7
        Textfield (250,275 100x30), "Bit 7"
    GroupBox (10,60 300x170), "Status Generic Instance"
        Textfield (180,30 50x30), "%s", text variable: DALI_Commissioning.fbPart300GenericDevice.nInputValue
        Textfield (180,70 50x30), "%s", text variable: DALI_Commissioning.fbPart300GenericDevice.nInstanceError
        Textfield (180,110 50x30), "%s", text variable: DALI_Commissioning.fbPart300GenericDevice.nResolution
        Textfield (10,30 160x30), "Input Value:"
        Textfield (10,70 160x30), "Instance Error:"
        Textfield (10,110 160x30), "Resolution:"
    Button (425,180 150x40), "Read"
        OnMouseClick: execute { DALI_Commissioning.fbPart300GenericDevice.bRead := TRUE; }
    WaitingSymbolFlower (360,200 70x70), invisible if: DALI_Commissioning.fbPart300GenericDevice.bHideWaitSymbol
    Button (595,180 150x40), "Write parameters"
        OnMouseClick: execute { DALI_Commissioning.fbPart300GenericDevice.bWrite := TRUE; }
    Textfield (425,130 150x40), "Instance Number:"
    Textfield (425,80 150x40), "Short Address:"
    Button (570,80 80x40), "%d", text variable: DALI_Commissioning.fbPart300GenericDevice.nAddress
        OnMouseClick: write the text variable via Default, min 0, max 63, title "Insert Short Address"
    Button (570,130 80x40), "%d", text variable: DALI_Commissioning.fbPart300GenericDevice.nInstanceAddress
        OnMouseClick: write the text variable via Default, min 0, max 31, title "Insert instance number"
    Group (10,5 170x40)
        Textfield (0,0 110x40), "DALI Line:"
        Button (90,0 80x40), "%d", text variable: GVL_Internal.nDALILine
            OnMouseClick: write the text variable via Default, min 1, max GVL_Internal.nNumberOfDALI_Lines, title "Choose line"
    Rectangle (332,37 150x30), "Identify"
        OnMouseDown: execute { DALI_Commissioning.fbPart300GenericDevice.bIdentify := TRUE; }
END_VISUALIZATION

// ---- Tc3_DALI_PLC_Commissioning_Tool/VISUs/Visu_DALICommissioning/Visu_Part301PushButton.TcVIS
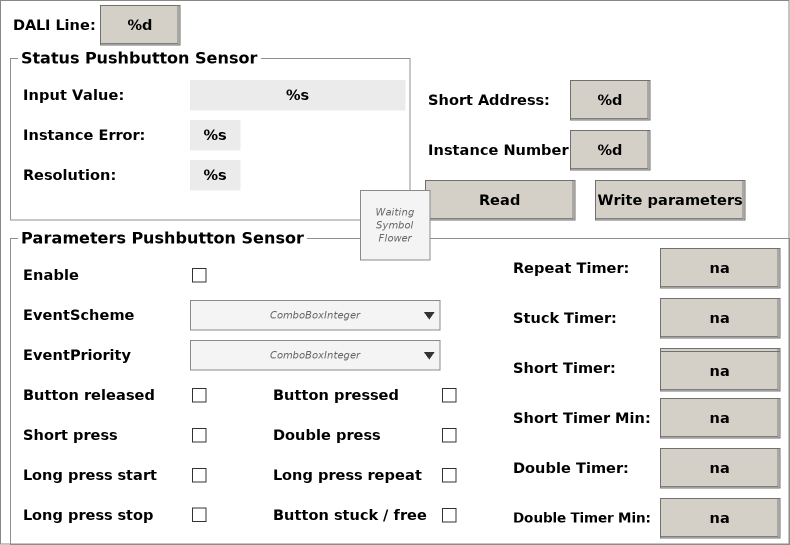
VISUALIZATION Visu_Part301PushButton  // 790x545
    GroupBox (10,230 780x315), "Parameters Pushbutton Sensor"
        Button (650,268 120x40), "%d ms", text variable: DALI_Commissioning.fbPart301PushButton.nDoubleMin
        Button (650,268 120x40), "na", invisible if: Not DALI_Commissioning.fbPart301PushButton.bNoDoubleTimer, input disabled if: Not DALI_Commissioning.fbPart301PushButton.bNoDoubleTimer
        Button (650,168 120x40), "%d ms", text variable: DALI_Commissioning.fbPart301PushButton.nShortMin
        Button (650,168 120x40), "na", invisible if: Not DALI_Commissioning.fbPart301PushButton.bNoRepeatTimer, input disabled if: Not DALI_Commissioning.fbPart301PushButton.bNoRepeatTimer
        Button (650,218 120x40), "%d ms", text variable: DALI_Commissioning.fbPart301PushButton.nDouble
            OnMouseClick: write the text variable via Default, min 0, max 2000, title "Insert value for double timer"
        Button (650,218 120x40), "na", invisible if: Not DALI_Commissioning.fbPart301PushButton.bNoDoubleTimer, input disabled if: Not DALI_Commissioning.fbPart301PushButton.bNoDoubleTimer
        Button (650,118 120x40), "%d ms", text variable: DALI_Commissioning.fbPart301PushButton.nShort
            OnMouseClick: write the text variable via Default, min 10, max 500, title "Insert value for short timer"
        Button (650,121 120x40), "na", invisible if: Not DALI_Commissioning.fbPart301PushButton.bNoRepeatTimer, input disabled if: Not DALI_Commissioning.fbPart301PushButton.bNoRepeatTimer
        Button (650,68 120x40), "%d s", text variable: DALI_Commissioning.fbPart301PushButton.nStuck
            OnMouseClick: write the text variable via Default, min 5, max 255, title "Insert value for stuck timer"
        Button (650,68 120x40), "na", invisible if: Not DALI_Commissioning.fbPart301PushButton.bNoRepeatTimer, input disabled if: Not DALI_Commissioning.fbPart301PushButton.bNoRepeatTimer
        Button (650,18 120x40), "%d ms", text variable: DALI_Commissioning.fbPart301PushButton.nRepeat
            OnMouseClick: write the text variable via Default, min 100, max 2000, title "Insert value for repeat timer"
        Button (650,18 120x40), "na", invisible if: Not DALI_Commissioning.fbPart301PushButton.bNoRepeatTimer, input disabled if: Not DALI_Commissioning.fbPart301PushButton.bNoRepeatTimer
        Textfield (500,23 145x30), "Repeat Timer:"
        Textfield (500,73 145x30), "Stuck Timer:"
        Textfield (500,123 145x30), "Short Timer:"
        Textfield (500,223 145x30), "Double Timer:"
        Textfield (10,30 170x30), "Enable"
        Checkbox (180,30 30x30), variable: DALI_Commissioning.fbPart301PushButton.bEnable
        Textfield (10,70 170x30), "EventScheme"
        Textfield (10,150 170x30), "Button released"
        Textfield (10,190 170x30), "Short press"
        Textfield (10,230 170x30), "Long press start"
        Textfield (10,270 170x30), "Long press stop"
        Textfield (260,150 170x30), "Button pressed"
        Textfield (260,190 170x30), "Double press"
        Textfield (260,230 170x30), "Long press repeat"
        Textfield (260,270 170x30), "Button stuck / free"
        Checkbox (180,150 30x30), variable: DALI_Commissioning.fbPart301PushButton.bButtonReleased
        Checkbox (180,190 30x30), variable: DALI_Commissioning.fbPart301PushButton.bShortPress
        Checkbox (180,230 30x30), variable: DALI_Commissioning.fbPart301PushButton.bLongPressStart
        Checkbox (430,150 30x30), variable: DALI_Commissioning.fbPart301PushButton.bButtonPressed
        Checkbox (430,190 30x30), variable: DALI_Commissioning.fbPart301PushButton.bDoublePress
        Checkbox (430,230 29x30), variable: DALI_Commissioning.fbPart301PushButton.bLongPressRepeat
        Checkbox (430,270 30x30), variable: DALI_Commissioning.fbPart301PushButton.bButtonStuck
        ComboBoxInteger (180,70 250x30), variable: DALI_Commissioning.fbPart301PushButton.eEventScheme, text list: 'EventScheme'
        Checkbox (180,270 28x29), variable: DALI_Commissioning.fbPart301PushButton.bLongPressStop
        Textfield (10,110 170x30), "EventPriority"
        ComboBoxInteger (180,110 250x30), variable: DALI_Commissioning.fbPart301PushButton.eEventPriority, text list: 'EventPriority'
        Textfield (500,173 145x30), "Short Timer Min:"
        Textfield (500,273 145x30), "Double Timer Min:"
    GroupBox (10,50 400x170), "Status Pushbutton Sensor"
        Textfield (10,30 160x30), "Input Value:"
        Textfield (10,70 160x30), "Instance Error:"
        Textfield (10,110 160x30), "Resolution:"
        Textfield (180,30 215x30), "%s", text variable: DALI_Commissioning.fbPart301PushButton.sInputValue
        Textfield (180,70 50x30), "%s", text variable: DALI_Commissioning.fbPart301PushButton.nInstanceError
        Textfield (180,110 50x30), "%s", text variable: DALI_Commissioning.fbPart301PushButton.nResolution
    Button (425,180 150x40), "Read"
        OnMouseClick: execute { DALI_Commissioning.fbPart301PushButton.bRead := TRUE; }
    WaitingSymbolFlower (360,190 70x70), invisible if: DALI_Commissioning.fbPart301PushButton.bHideWaitSymbol
    Button (595,180 150x40), "Write parameters"
        OnMouseClick: execute { DALI_Commissioning.fbPart301PushButton.bWrite := TRUE; }
    Group (10,5 170x40)
        Textfield (0,0 110x40), "DALI Line:"
        Button (90,0 80x40), "%d", text variable: GVL_Internal.nDALILine
            OnMouseClick: write the text variable via Default, min 1, max GVL_Internal.nNumberOfDALI_Lines, title "Choose line"
    Textfield (425,80 160x40), "Short Address:"
    Button (570,80 80x40), "%d", text variable: DALI_Commissioning.fbPart301PushButton.nAddress
        OnMouseClick: write the text variable via Default, min 0, max 63, title "Insert Short Address"
    Textfield (425,130 150x40), "Instance Number:"
    Button (570,130 80x40), "%d", text variable: DALI_Commissioning.fbPart301PushButton.nInstanceAddress
        OnMouseClick: write the text variable via Default, min 0, max 31, title "Insert instance number"
END_VISUALIZATION

// ---- Tc3_DALI_PLC_Commissioning_Tool/VISUs/Visu_DALICommissioning/Visu_Part302AbsoluteInputDevice.TcVIS
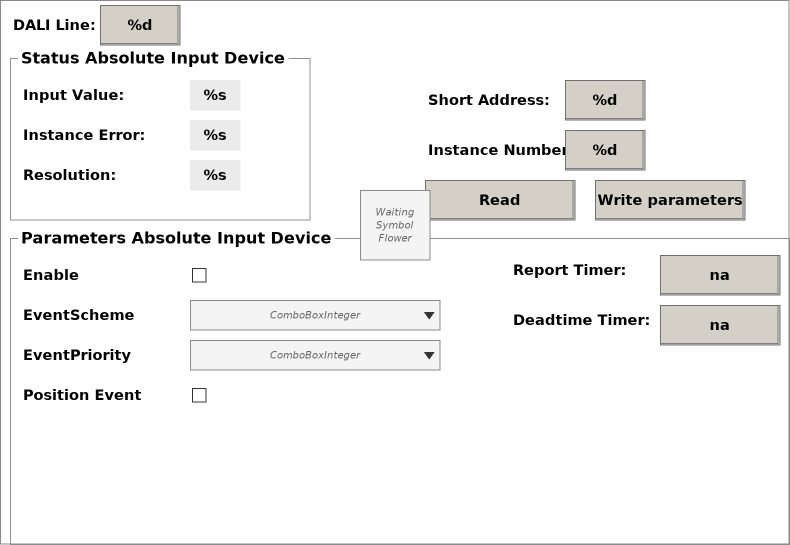
VISUALIZATION Visu_Part302AbsoluteInputDevice  // 790x545
    GroupBox (10,50 300x170), "Status Absolute Input Device"
        Textfield (10,30 160x30), "Input Value:"
        Textfield (10,70 160x30), "Instance Error:"
        Textfield (10,110 160x30), "Resolution:"
        Textfield (180,30 50x30), "%s", text variable: DALI_Commissioning.fbPart302AbsoluteInputDevice.nInputValue
        Textfield (180,70 50x30), "%s", text variable: DALI_Commissioning.fbPart302AbsoluteInputDevice.nInstanceError
        Textfield (180,110 50x30), "%s", text variable: DALI_Commissioning.fbPart302AbsoluteInputDevice.nResolution
    Button (425,180 150x40), "Read"
        OnMouseClick: execute { DALI_Commissioning.fbPart302AbsoluteInputDevice.bRead := TRUE; }
    GroupBox (10,230 780x315), "Parameters Absolute Input Device"
        Textfield (500,75 145x30), "Deadtime Timer:"
        Textfield (500,25 145x30), "Report Timer:"
        Textfield (10,30 150x30), "Enable"
        Button (650,25 120x40), "%d s", text variable: DALI_Commissioning.fbPart302AbsoluteInputDevice.nReport
            OnMouseClick: write DALI_Commissioning.fbPart302AbsoluteInputDevice.nReport via Default, min 0, max 255, title "Insert value for report timer"
        Button (650,75 120x40), "%d ms", text variable: DALI_Commissioning.fbPart302AbsoluteInputDevice.nDeadtime
            OnMouseClick: write DALI_Commissioning.fbPart302AbsoluteInputDevice.nDeadtime via Default, min 0, max 12750, title "Insert value for deadtime timer"
        Checkbox (180,30 30x30), variable: DALI_Commissioning.fbPart302AbsoluteInputDevice.bEnable
        Textfield (10,70 150x30), "EventScheme"
        ComboBoxInteger (180,70 250x30), variable: DALI_Commissioning.fbPart302AbsoluteInputDevice.eEventScheme, text list: 'EventScheme'
        Button (650,25 120x40), "na", invisible if: Not DALI_Commissioning.fbPart302AbsoluteInputDevice.bNoReportTimer, input disabled if: Not DALI_Commissioning.fbPart302AbsoluteInputDevice.bNoReportTimer
        Button (650,75 120x40), "na", invisible if: Not DALI_Commissioning.fbPart302AbsoluteInputDevice.bNoDeadtimeTimer, input disabled if: Not DALI_Commissioning.fbPart302AbsoluteInputDevice.bNoDeadtimeTimer
        Textfield (10,110 150x30), "EventPriority"
        Textfield (10,150 150x30), "Position Event"
        ComboBoxInteger (180,110 250x30), variable: DALI_Commissioning.fbPart302AbsoluteInputDevice.eEventPriority, text list: 'EventPriority'
        Checkbox (180,150 30x30), variable: DALI_Commissioning.fbPart302AbsoluteInputDevice.bPositionEventEnabled
    WaitingSymbolFlower (360,190 70x70), invisible if: DALI_Commissioning.fbPart302AbsoluteInputDevice.bHideWaitSymbol
    Button (595,180 150x40), "Write parameters"
        OnMouseClick: execute { DALI_Commissioning.fbPart302AbsoluteInputDevice.bWrite := TRUE; }
    Group (10,5 170x40)
        Textfield (0,0 110x40), "DALI Line:"
        Button (90,0 80x40), "%d", text variable: GVL_Internal.nDALILine
            OnMouseClick: write the text variable via Default, min 1, max GVL_Internal.nNumberOfDALI_Lines, title "Choose line"
    Textfield (425,80 130x40), "Short Address:"
    Button (565,80 80x40), "%d", text variable: DALI_Commissioning.fbPart302AbsoluteInputDevice.nAddress
        OnMouseClick: write DALI_Commissioning.fbPart302AbsoluteInputDevice.nAddress via Default, min 0, max 63, title "Insert Short Address"
    Textfield (425,130 150x40), "Instance Number:"
    Button (565,130 80x40), "%d", text variable: DALI_Commissioning.fbPart302AbsoluteInputDevice.nInstanceAddress
        OnMouseClick: write DALI_Commissioning.fbPart302AbsoluteInputDevice.nInstanceAddress via Default, min 0, max 31, title "Insert instance number"
END_VISUALIZATION

// ---- Tc3_DALI_PLC_Commissioning_Tool/VISUs/Visu_DALICommissioning/Visu_Part303OccupancySensor.TcVIS
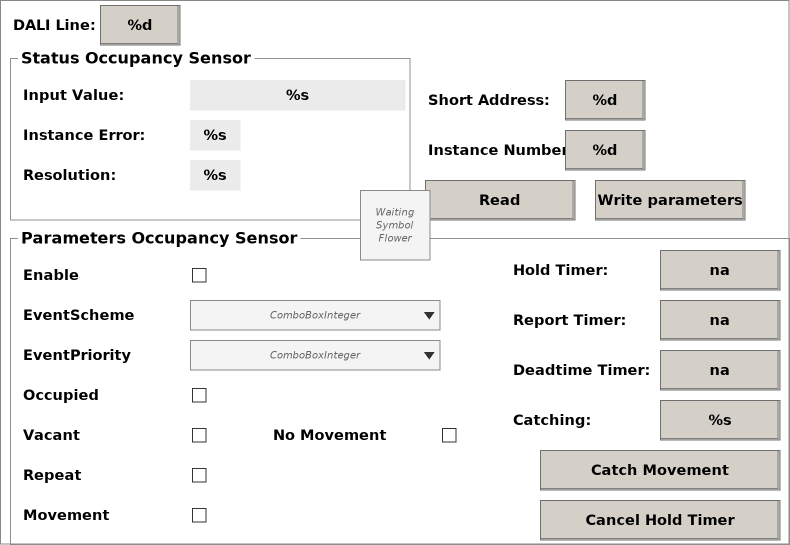
VISUALIZATION Visu_Part303OccupancySensor  // 790x545
    GroupBox (10,230 780x315), "Parameters Occupancy Sensor"
        Button (650,70 120x40), "%d s", text variable: DALI_Commissioning.fbPart303OccupancySensor.nReport
            OnMouseClick: write the text variable via Default, min 0, max 255, title "Insert value for report timer"
        Button (650,70 120x40), "na", invisible if: Not DALI_Commissioning.fbPart303OccupancySensor.bNoReportTimer, input disabled if: Not DALI_Commissioning.fbPart303OccupancySensor.bNoReportTimer
        Textfield (500,125 145x30), "Deadtime Timer:"
        Textfield (500,75 145x30), "Report Timer:"
        Textfield (500,25 145x30), "Hold Timer:"
        Button (650,20 120x40), "%d s", text variable: DALI_Commissioning.fbPart303OccupancySensor.nHold, invisible if: DALI_Commissioning.fbPart303OccupancySensor.bNoHoldTimer, input disabled if: DALI_Commissioning.fbPart303OccupancySensor.bNoHoldTimer
            OnMouseClick: write the text variable via Default, min 0, max 2538, title "Insert value for hold timer"
        Textfield (10,30 150x30), "Enable"
        Button (650,120 120x40), "%d ms", text variable: DALI_Commissioning.fbPart303OccupancySensor.nDeadtime
            OnMouseClick: write the text variable via Default, min 0, max 12750, title "Insert value for deadtime timer"
        Checkbox (180,30 30x30), variable: DALI_Commissioning.fbPart303OccupancySensor.bEnable
        Textfield (10,70 150x30), "EventScheme"
        Textfield (10,150 150x30), "Occupied"
        Textfield (10,190 150x30), "Vacant"
        Textfield (10,230 150x30), "Repeat"
        Textfield (10,270 150x30), "Movement"
        Textfield (260,190 150x30), "No Movement"
        Checkbox (180,150 30x30), variable: DALI_Commissioning.fbPart303OccupancySensor.bOccupied
        Checkbox (180,190 30x30), variable: DALI_Commissioning.fbPart303OccupancySensor.bVacant
        Checkbox (180,230 30x30), variable: DALI_Commissioning.fbPart303OccupancySensor.bRepeat
        Checkbox (430,190 30x30), variable: DALI_Commissioning.fbPart303OccupancySensor.bNoMovement
        ComboBoxInteger (180,70 250x30), variable: DALI_Commissioning.fbPart303OccupancySensor.eEventScheme, text list: 'EventScheme'
        Checkbox (180,270 30x30), variable: DALI_Commissioning.fbPart303OccupancySensor.bMovement
        Button (650,120 120x40), "na", invisible if: Not DALI_Commissioning.fbPart303OccupancySensor.bNoDeadtimeTimer, input disabled if: Not DALI_Commissioning.fbPart303OccupancySensor.bNoDeadtimeTimer
        Button (530,270 240x40), "Cancel Hold Timer"
            OnMouseClick: execute { DALI_Commissioning.fbPart303OccupancySensor.bCancelHoldTimer := true; }
        Textfield (10,110 150x30), "EventPriority"
        ComboBoxInteger (180,110 250x30), variable: DALI_Commissioning.fbPart303OccupancySensor.eEventPriority, text list: 'EventPriority'
        Button (650,20 120x40), "na", invisible if: Not DALI_Commissioning.fbPart303OccupancySensor.bNoHoldTimer, input disabled if: Not DALI_Commissioning.fbPart303OccupancySensor.bNoHoldTimer
        Button (530,220 240x40), "Catch Movement"
            OnMouseClick: execute { DALI_Commissioning.fbPart303OccupancySensor.bCatchMovement := true; }
        Textfield (500,175 145x30), "Catching:"
    GroupBox (10,50 400x170), "Status Occupancy Sensor"
        Textfield (10,30 160x30), "Input Value:"
        Textfield (10,70 160x30), "Instance Error:"
        Textfield (10,110 160x30), "Resolution:"
        Textfield (180,30 215x30), "%s", text variable: DALI_Commissioning.fbPart303OccupancySensor.sInputValue
        Textfield (180,70 50x30), "%s", text variable: DALI_Commissioning.fbPart303OccupancySensor.nInstanceError
        Textfield (180,110 50x30), "%s", text variable: DALI_Commissioning.fbPart303OccupancySensor.nResolution
    Button (425,180 150x40), "Read"
        OnMouseClick: execute { DALI_Commissioning.fbPart303OccupancySensor.bRead := TRUE; }
    WaitingSymbolFlower (360,190 70x70), invisible if: DALI_Commissioning.fbPart303OccupancySensor.bHideWaitSymbol
    Button (595,180 150x40), "Write parameters"
        OnMouseClick: execute { DALI_Commissioning.fbPart303OccupancySensor.bWrite := TRUE; }
    Button (660,400 120x40), "%s", text variable: DALI_Commissioning.fbPart303OccupancySensor.sCatching
        OnMouseClick: write the text variable via Default, min 0, max 12750, title "Insert value for deadtime timer"
    Group (10,5 170x40)
        Textfield (0,0 110x40), "DALI Line:"
        Button (90,0 80x40), "%d", text variable: GVL_Internal.nDALILine
            OnMouseClick: write the text variable via Default, min 1, max GVL_Internal.nNumberOfDALI_Lines, title "Choose line"
    Textfield (425,80 130x40), "Short Address:"
    Button (565,80 80x40), "%d", text variable: DALI_Commissioning.fbPart303OccupancySensor.nAddress
        OnMouseClick: write the text variable via Default, min 0, max 63, title "Insert Short Address"
    Textfield (425,130 150x40), "Instance Number:"
    Button (565,130 80x40), "%d", text variable: DALI_Commissioning.fbPart303OccupancySensor.nInstanceAddress
        OnMouseClick: write the text variable via Default, min 0, max 31, title "Insert instance number"
END_VISUALIZATION

// ---- Tc3_DALI_PLC_Commissioning_Tool/VISUs/Visu_DALICommissioning/Visu_Part304LightSensor.TcVIS
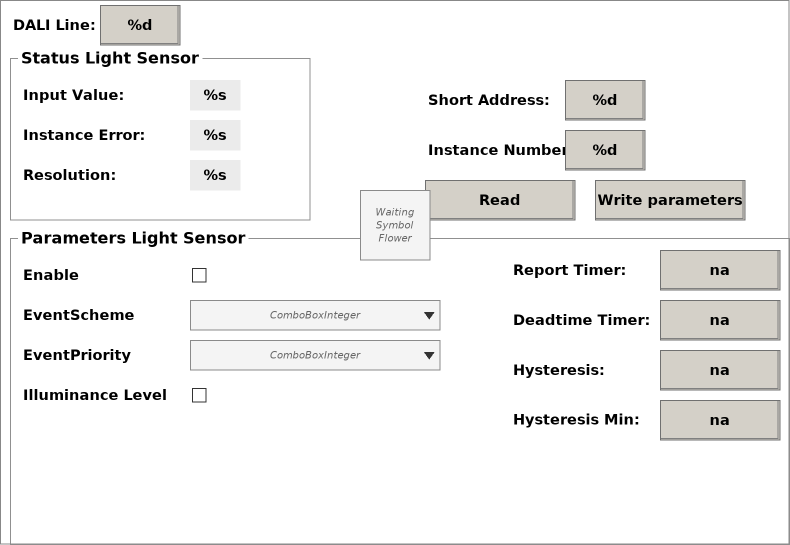
VISUALIZATION Visu_Part304LightSensor  // 790x545
    GroupBox (10,230 780x315), "Parameters Light Sensor"
        Button (650,170 120x40), "%d", text variable: DALI_Commissioning.fbPart304LightSensor.nHysteresisMin
            OnMouseClick: write the text variable via Default, min 0, max 255, title "Insert value for hysteresis min"
        Button (650,170 120x40), "na", invisible if: not DALI_Commissioning.fbPart304LightSensor.bNoHysteresisMin, input disabled if: not DALI_Commissioning.fbPart304LightSensor.bNoHysteresisMin
        Button (650,20 120x40), "%d s", text variable: DALI_Commissioning.fbPart304LightSensor.nReport
            OnMouseClick: write the text variable via Default, min 0, max 255, title "Insert value for report timer"
        Button (650,70 120x40), "%d ms", text variable: DALI_Commissioning.fbPart304LightSensor.nDeadtime
            OnMouseClick: write the text variable via Default, min 0, max 12750, title "Insert value for deadtime timer"
        Button (650,120 120x40), "%d %", text variable: DALI_Commissioning.fbPart304LightSensor.nHysteresis
            OnMouseClick: write the text variable via Default, min 0, max 25, title "Insert value for hysteresis"
        Button (650,120 120x40), "na", invisible if: not DALI_Commissioning.fbPart304LightSensor.bNoHysteresis, input disabled if: not DALI_Commissioning.fbPart304LightSensor.bNoHysteresis
        Button (650,70 120x40), "na", invisible if: not DALI_Commissioning.fbPart304LightSensor.bNoDeadtimeTimer, input disabled if: not DALI_Commissioning.fbPart304LightSensor.bNoDeadtimeTimer
        Button (650,20 120x40), "na", invisible if: not DALI_Commissioning.fbPart304LightSensor.bNoReportTimer, input disabled if: not DALI_Commissioning.fbPart304LightSensor.bNoReportTimer
        Textfield (500,175 145x29), "Hysteresis Min:"
        Textfield (500,125 145x30), "Hysteresis:"
        Textfield (500,25 145x30), "Report Timer:"
        Textfield (500,75 145x30), "Deadtime Timer:"
        Textfield (10,30 150x30), "Enable"
        Checkbox (180,30 30x30), variable: DALI_Commissioning.fbPart304LightSensor.bEnable
        Textfield (10,70 150x30), "EventScheme"
        Textfield (10,150 150x30), "Illuminance Level"
        ComboBoxInteger (180,70 250x30), variable: DALI_Commissioning.fbPart304LightSensor.eEventScheme, text list: 'EventScheme'
        Checkbox (180,150 30x30), variable: DALI_Commissioning.fbPart304LightSensor.bIlluminanceLevel
        Textfield (10,110 150x30), "EventPriority"
        ComboBoxInteger (180,110 250x30), variable: DALI_Commissioning.fbPart304LightSensor.eEventPriority, text list: 'EventPriority'
    GroupBox (10,50 300x170), "Status Light Sensor"
        Textfield (10,30 160x30), "Input Value:"
        Textfield (10,70 160x30), "Instance Error:"
        Textfield (10,110 160x30), "Resolution:"
        Textfield (180,30 50x30), "%s", text variable: DALI_Commissioning.fbPart304LightSensor.nInputValue
        Textfield (180,70 50x30), "%s", text variable: DALI_Commissioning.fbPart304LightSensor.nInstanceError
        Textfield (180,110 50x30), "%s", text variable: DALI_Commissioning.fbPart304LightSensor.nResolution
    Button (425,180 150x40), "Read"
        OnMouseClick: execute { DALI_Commissioning.fbPart304LightSensor.bRead := TRUE; }
    WaitingSymbolFlower (360,190 70x70), invisible if: DALI_Commissioning.fbPart304LightSensor.bHideWaitSymbol
    Button (595,180 150x40), "Write parameters"
        OnMouseClick: execute { DALI_Commissioning.fbPart304LightSensor.bWrite := TRUE; }
    Textfield (425,80 130x40), "Short Address:"
    Button (565,80 80x40), "%d", text variable: DALI_Commissioning.fbPart304LightSensor.nAddress
        OnMouseClick: write the text variable via Default, min 0, max 63, title "Insert Short Address"
    Textfield (425,130 150x40), "Instance Number:"
    Button (565,130 80x40), "%d", text variable: DALI_Commissioning.fbPart304LightSensor.nInstanceAddress
        OnMouseClick: write the text variable via Default, min 0, max 31, title "Insert instance number"
    Group (10,5 170x40)
        Textfield (0,0 110x40), "DALI Line:"
        Button (90,0 80x40), "%d", text variable: GVL_Internal.nDALILine
            OnMouseClick: write the text variable via Default, min 1, max GVL_Internal.nNumberOfDALI_Lines, title "Choose line"
END_VISUALIZATION
